TYPE ST_Msg_PTP :
STRUCT
	targetJoint : ARRAY[1..6] OF LREAL;
	executeTime : LREAL;
	cycles : USINT;  
END_STRUCT
END_TYPE

(* stored: Version 1.1.0.1, ProductVersion 3.1.4024.12
   DUT ST_Msg_PTP: Id {c3a67d99-3ec8-425f-a9c4-b2388ca808fe} *)
